REGION Network 53: Immediate Stop
   RUNG wire#powerrail
      { S7_Templates := "SrcType := DInt" } EQ_Contact(in1 := "Unit1.Em8.ControlNodes".hipotThickness.sequence.status.currentStep, in2 := #STEP_IMMEDIATE_STOP)
      Contact( "Unit1.Em8.ControlNodes".hipotThickness.sequence.status.seqActive )
      wire#w1
      I_Contact( "Unit1.Em8.ControlNodes".hipotThickness."step".transition1[9999] )
      Coil( "Unit1.Em8.ControlNodes".hipotThickness."step".action1[9999] )
   END_RUNG
   RUNG wire#w1
      Contact( "Unit1.Em8.ControlNodes".hipotThickness."step".action1[9999] )
      Coil( "Unit1.Em8.ControlNodes".hipotThickness."step".transition1[9999] )
   END_RUNG
   RUNG wire#w1
      Contact( "Unit1.Em8.ControlNodes".hipotThickness."step".transition1[9999] )
      Coil( #tempDo_nothing_and_wait_for_init )
   END_RUNG
   // the same network as SCL:
   #_w1 := ("Unit1.Em8.ControlNodes".hipotThickness.sequence.status.currentStep = #STEP_IMMEDIATE_STOP) AND "Unit1.Em8.ControlNodes".hipotThickness.sequence.status.seqActive;
   "Unit1.Em8.ControlNodes".hipotThickness."step".action1[9999] := #_w1 AND NOT "Unit1.Em8.ControlNodes".hipotThickness."step".transition1[9999];
   "Unit1.Em8.ControlNodes".hipotThickness."step".transition1[9999] := #_w1 AND "Unit1.Em8.ControlNodes".hipotThickness."step".action1[9999];
   #tempDo_nothing_and_wait_for_init := #_w1 AND "Unit1.Em8.ControlNodes".hipotThickness."step".transition1[9999];
END_REGION

REGION Network 54: ********************** STATUS **************************
END_REGION

REGION Network 55: Sequence Status
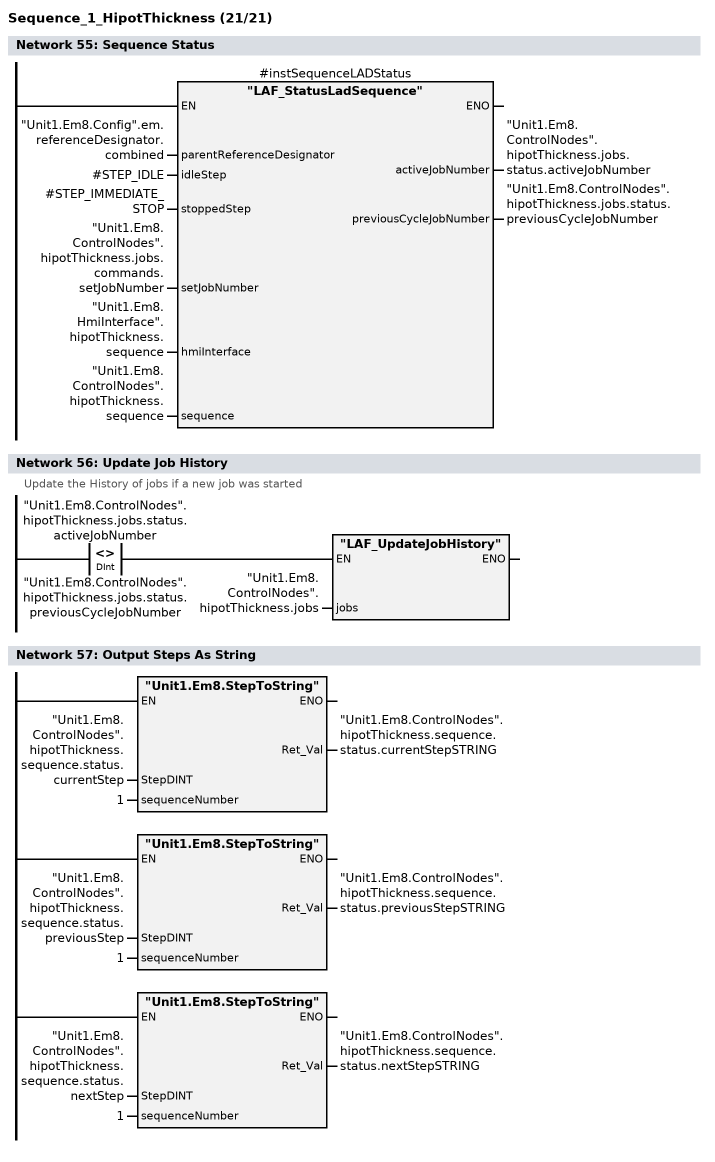
   RUNG wire#powerrail
      #instSequenceLADStatus(parentReferenceDesignator := "Unit1.Em8.Config".em.referenceDesignator.combined, idleStep := #STEP_IDLE, stoppedStep := #STEP_IMMEDIATE_STOP, setJobNumber := "Unit1.Em8.ControlNodes".hipotThickness.jobs.commands.setJobNumber, hmiInterface := "Unit1.Em8.HmiInterface".hipotThickness.sequence, sequence := "Unit1.Em8.ControlNodes".hipotThickness.sequence, activeJobNumber => "Unit1.Em8.ControlNodes".hipotThickness.jobs.status.activeJobNumber, previousCycleJobNumber => "Unit1.Em8.ControlNodes".hipotThickness.jobs.status.previousCycleJobNumber)
   END_RUNG
   // the same network as SCL:
   #instSequenceLADStatus(parentReferenceDesignator := "Unit1.Em8.Config".em.referenceDesignator.combined,   // "LAF_StatusLadSequence"
                          idleStep := #STEP_IDLE,
                          stoppedStep := #STEP_IMMEDIATE_STOP,
                          setJobNumber := "Unit1.Em8.ControlNodes".hipotThickness.jobs.commands.setJobNumber,
                          hmiInterface := "Unit1.Em8.HmiInterface".hipotThickness.sequence,
                          sequence := "Unit1.Em8.ControlNodes".hipotThickness.sequence,
                          activeJobNumber => "Unit1.Em8.ControlNodes".hipotThickness.jobs.status.activeJobNumber,
                          previousCycleJobNumber => "Unit1.Em8.ControlNodes".hipotThickness.jobs.status.previousCycleJobNumber);
END_REGION

REGION Network 56: Update Job History
   // Update the History of jobs if a new job was started
   RUNG wire#powerrail
      { S7_Templates := "SrcType := DInt" } NE_Contact(in1 := "Unit1.Em8.ControlNodes".hipotThickness.jobs.status.activeJobNumber, in2 := "Unit1.Em8.ControlNodes".hipotThickness.jobs.status.previousCycleJobNumber)
      "LAF_UpdateJobHistory"(jobs := "Unit1.Em8.ControlNodes".hipotThickness.jobs)
   END_RUNG
   // the same network as SCL:
   IF "Unit1.Em8.ControlNodes".hipotThickness.jobs.status.activeJobNumber <> "Unit1.Em8.ControlNodes".hipotThickness.jobs.status.previousCycleJobNumber THEN
       "LAF_UpdateJobHistory"(jobs := "Unit1.Em8.ControlNodes".hipotThickness.jobs);
   END_IF;
END_REGION

REGION Network 57: Output Steps As String
   RUNG wire#powerrail
      "Unit1.Em8.StepToString"(StepDINT := "Unit1.Em8.ControlNodes".hipotThickness.sequence.status.currentStep, sequenceNumber := 1, Ret_Val => "Unit1.Em8.ControlNodes".hipotThickness.sequence.status.currentStepSTRING)
   END_RUNG
   RUNG wire#powerrail
      "Unit1.Em8.StepToString"(StepDINT := "Unit1.Em8.ControlNodes".hipotThickness.sequence.status.previousStep, sequenceNumber := 1, Ret_Val => "Unit1.Em8.ControlNodes".hipotThickness.sequence.status.previousStepSTRING)
   END_RUNG
   RUNG wire#powerrail
      "Unit1.Em8.StepToString"(StepDINT := "Unit1.Em8.ControlNodes".hipotThickness.sequence.status.nextStep, sequenceNumber := 1, Ret_Val => "Unit1.Em8.ControlNodes".hipotThickness.sequence.status.nextStepSTRING)
   END_RUNG
   // the same network as SCL:
   "Unit1.Em8.ControlNodes".hipotThickness.sequence.status.currentStepSTRING := "Unit1.Em8.StepToString"(StepDINT := "Unit1.Em8.ControlNodes".hipotThickness.sequence.status.currentStep,
                           sequenceNumber := 1);
   "Unit1.Em8.ControlNodes".hipotThickness.sequence.status.previousStepSTRING := "Unit1.Em8.StepToString"(StepDINT := "Unit1.Em8.ControlNodes".hipotThickness.sequence.status.previousStep,
                           sequenceNumber := 1);
   "Unit1.Em8.ControlNodes".hipotThickness.sequence.status.nextStepSTRING := "Unit1.Em8.StepToString"(StepDINT := "Unit1.Em8.ControlNodes".hipotThickness.sequence.status.nextStep,
                           sequenceNumber := 1);
END_REGION
END_FUNCTION_BLOCK
